FUNCTION_BLOCK CustomStateCommand EXTENDS CommandBase
VAR_INPUT
END_VAR
VAR_OUTPUT
END_VAR
VAR
	fbDelayedState: TON := (IN := FALSE, PT:= T#2S);
END_VAR

// OO-Class 
SUPER^();

// Will be called when ``stHandshake.bExecute`` changes to ``true`` one cycle and in the same cycle.
METHOD PROTECTED Init
VAR_INPUT
END_VAR
fbDelayedState(IN := False);
END_METHOD

// Execute the funktional part of the command implementation. Will also be executed in the same cycle ``stHandshake.bExecute`` changes to ``true`` after the ``Init`` Method
METHOD PROTECTED Task : BOOL

fbDelayedState(IN:= TRUE);

IF (fbDelayedState.Q) THEN
	Finish(E_CommandResultCode.StartCustom + 1);
END_IF
END_METHOD

END_FUNCTION_BLOCK

(* stored: Version 1.1.0.1, ProductVersion 3.1.4022.10
   POU CustomStateCommand: Id {096afba5-ac69-0cc5-0827-85acbc768d34}, SpecialFunc None
   Method Init: Id {3e6108ad-08e0-04ed-2de4-0e3f0a82760a}
   Method Task: Id {43834ce9-c5dd-03ca-0d2d-226e73644be2} *)
